{attribute 'linkalways'} 
FUNCTION GetByteOffset : PVOID
VAR_INPUT
	Structure : ANY;
	Member : ANY_BIT; 
END_VAR

GetByteOffset := Member.pValue - Structure.pValue;

END_FUNCTION

(* stored: Version 1.1.0.1, ProductVersion 3.1.4024.12
   POU GetByteOffset: Id {a67859da-19f3-4eec-96e6-e9fe3265bb09}, SpecialFunc None *)
